# EPICS substitutions: modules/event/evrSupport/Db/ioc/IOC-IN20-PM05evr.substitutions
#==============================================================================
#
# Abs:  LCLS EVR IOC records for IN20 PM05
#
# Name: IOC-IN20-PM05evr.substitutions
#
#==============================================================================
#
file evrPMXX.db
{
pattern { DEVICE        }
	{ EVR:IN20:PM05 }
}
